Staubli VAL3: setTool.pgx

public program setTool(tool x_tTool, num x_nIndex)
begin
  // define the tool
  saveData:tData[x_nIndex].tcp=flange
  saveData:tData[x_nIndex].tcp.trsf=x_tTool.trsf
  saveData:tData[x_nIndex].tcp.ctime=x_tTool.ctime
  saveData:tData[x_nIndex].tcp.otime=x_tTool.otime
end
